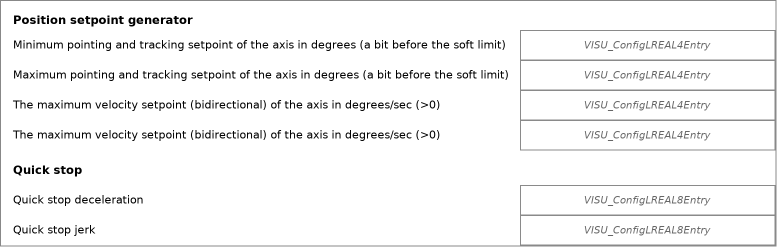
VISUALIZATION VISU_AxesConfig_Rotation_2  // 777x247
VAR_IN_OUT
    active : AxesRotationConfig;
    editable : AxesRotationConfig;
END_VAR
    Label (10,5 205x30), "Position setpoint generator"
    Label (10,30 495x30), "Minimum pointing and tracking setpoint of the axis in degrees (a bit before the soft limit)"
    Label (10,60 510x30), "Maximum pointing and tracking setpoint of the axis in degrees (a bit before the soft limit)"
    Label (10,90 475x30), "The maximum velocity setpoint (bidirectional) of the axis in degrees/sec (>0)"
    Label (10,120 475x30), "The maximum velocity setpoint (bidirectional) of the axis in degrees/sec (>0)"
    Frame (520,30 255x30)
        shows VISU_ConfigLREAL4Entry(active := active.minPositionSetpoint, editable := editable.minPositionSetpoint)
    Frame (520,60 255x30)
        shows VISU_ConfigLREAL4Entry(active := active.maxPositionSetpoint, editable := editable.maxPositionSetpoint)
    Frame (520,90 255x30)
        shows VISU_ConfigLREAL4Entry(active := active.maxVelocitySetpoint, editable := editable.maxVelocitySetpoint)
    Frame (520,120 255x30)
        shows VISU_ConfigLREAL4Entry(active := active.maxAccelerationSetpoint, editable := editable.maxAccelerationSetpoint)
    Label (10,155 205x30), "Quick stop"
    Frame (520,185 255x30)
        shows VISU_ConfigLREAL8Entry(active := active.quickStopDeceleration, editable := editable.quickStopDeceleration)
    Label (10,185 500x30), "Quick stop deceleration"
    Label (10,215 500x30), "Quick stop jerk"
    Frame (520,215 255x30)
        shows VISU_ConfigLREAL8Entry(active := active.quickStopJerk, editable := editable.quickStopJerk)
END_VISUALIZATION

(* stored: Version 1.1.0.1, ProductVersion 3.1.4019.2
   Visu VISU_AxesConfig_Rotation_2: Id {aa6e8c5b-56d9-402b-91d7-231a63f7c84b} *)
